# EPICS alarm handler configuration: alh_files/mgnt_li28_lgps.alhConfig
GROUP NULL LGPS:LI28:MG01
$ALIAS LGPS
$GUIDANCE
LI28 LGPS magnets
   Group Name: LGPS:LI28:MG01
   Summary PV:  LGPS:LI28:MG01:STATSUMY
$END

GROUP LGPS:LI28:MG01  LGPS:LI28:2
CHANNEL     LGPS:LI28:2           LGPS:LI28:2:STATMSG   -----
   $FORCEPV LGPS:LI28:2:STATMSGSV -DATL 1 0
